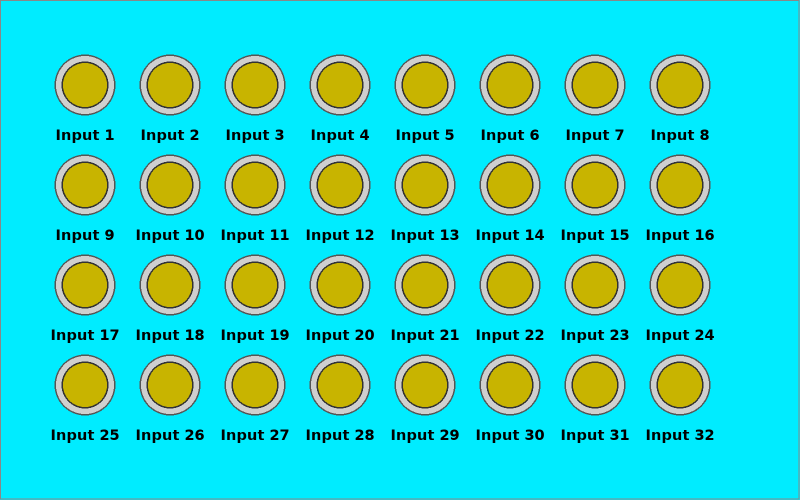
VISUALIZATION Screen_1_Sub_2  // 800x500
    Rectangle (0,0 800x500)
    Lamp1 (50,50 70x70), tooltip "Lamp 1", variable: GVL.HMI_Display_Lamp[0], style: Lamp-Lamp1-Yellow
    Label (50,120 70x30), "Input 1"
    Lamp1 (50,150 70x70), tooltip "Lamp 1", variable: GVL.HMI_Display_Lamp[8], style: Lamp-Lamp1-Yellow
    Label (50,220 70x30), "Input 9"
    Lamp1 (50,250 70x70), tooltip "Lamp 1", variable: GVL.HMI_Display_Lamp[16], style: Lamp-Lamp1-Yellow
    Label (50,320 70x30), "Input 17"
    Lamp1 (50,350 70x70), tooltip "Lamp 1", variable: GVL.HMI_Display_Lamp[24], style: Lamp-Lamp1-Yellow
    Label (50,420 70x30), "Input 25"
    Lamp1 (135,50 70x70), tooltip "Lamp 1", variable: GVL.HMI_Display_Lamp[1], style: Lamp-Lamp1-Yellow
    Label (135,120 70x30), "Input 2"
    Lamp1 (135,150 70x70), tooltip "Lamp 1", variable: GVL.HMI_Display_Lamp[9], style: Lamp-Lamp1-Yellow
    Label (135,220 70x30), "Input 10"
    Lamp1 (135,250 70x70), tooltip "Lamp 1", variable: GVL.HMI_Display_Lamp[17], style: Lamp-Lamp1-Yellow
    Label (135,320 70x30), "Input 18"
    Lamp1 (135,350 70x70), tooltip "Lamp 1", variable: GVL.HMI_Display_Lamp[25], style: Lamp-Lamp1-Yellow
    Label (135,420 70x30), "Input 26"
    Lamp1 (220,50 70x70), tooltip "Lamp 1", variable: GVL.HMI_Display_Lamp[2], style: Lamp-Lamp1-Yellow
    Label (220,120 70x30), "Input 3"
    Lamp1 (220,150 70x70), tooltip "Lamp 1", variable: GVL.HMI_Display_Lamp[10], style: Lamp-Lamp1-Yellow
    Label (220,220 70x30), "Input 11"
    Lamp1 (220,250 70x70), tooltip "Lamp 1", variable: GVL.HMI_Display_Lamp[18], style: Lamp-Lamp1-Yellow
    Label (220,320 70x30), "Input 19"
    Lamp1 (220,350 70x70), tooltip "Lamp 1", variable: GVL.HMI_Display_Lamp[26], style: Lamp-Lamp1-Yellow
    Label (220,420 70x30), "Input 27"
    Lamp1 (305,50 70x70), tooltip "Lamp 1", variable: GVL.HMI_Display_Lamp[3], style: Lamp-Lamp1-Yellow
    Label (305,120 70x30), "Input 4"
    Lamp1 (305,150 70x70), tooltip "Lamp 1", variable: GVL.HMI_Display_Lamp[11], style: Lamp-Lamp1-Yellow
    Label (305,220 70x30), "Input 12"
    Lamp1 (305,250 70x70), tooltip "Lamp 1", variable: GVL.HMI_Display_Lamp[19], style: Lamp-Lamp1-Yellow
    Label (305,320 70x30), "Input 20"
    Lamp1 (305,350 70x70), tooltip "Lamp 1", variable: GVL.HMI_Display_Lamp[27], style: Lamp-Lamp1-Yellow
    Label (305,420 70x30), "Input 28"
    Lamp1 (390,50 70x70), tooltip "Lamp 1", variable: GVL.HMI_Display_Lamp[4], style: Lamp-Lamp1-Yellow
    Label (390,120 70x30), "Input 5"
    Lamp1 (390,150 70x70), tooltip "Lamp 1", variable: GVL.HMI_Display_Lamp[12], style: Lamp-Lamp1-Yellow
    Label (390,220 70x30), "Input 13"
    Lamp1 (390,250 70x70), tooltip "Lamp 1", variable: GVL.HMI_Display_Lamp[20], style: Lamp-Lamp1-Yellow
    Label (390,320 70x30), "Input 21"
    Lamp1 (390,350 70x70), tooltip "Lamp 1", variable: GVL.HMI_Display_Lamp[28], style: Lamp-Lamp1-Yellow
    Label (390,420 70x30), "Input 29"
    Lamp1 (475,50 70x70), tooltip "Lamp 1", variable: GVL.HMI_Display_Lamp[5], style: Lamp-Lamp1-Yellow
    Label (475,120 70x30), "Input 6"
    Lamp1 (475,150 70x70), tooltip "Lamp 1", variable: GVL.HMI_Display_Lamp[13], style: Lamp-Lamp1-Yellow
    Label (475,220 70x30), "Input 14"
    Lamp1 (475,250 70x70), tooltip "Lamp 1", variable: GVL.HMI_Display_Lamp[21], style: Lamp-Lamp1-Yellow
    Label (475,320 70x30), "Input 22"
    Lamp1 (475,350 70x70), tooltip "Lamp 1", variable: GVL.HMI_Display_Lamp[29], style: Lamp-Lamp1-Yellow
    Label (475,420 70x30), "Input 30"
    Lamp1 (560,50 70x70), tooltip "Lamp 1", variable: GVL.HMI_Display_Lamp[6], style: Lamp-Lamp1-Yellow
    Label (560,120 70x30), "Input 7"
    Lamp1 (560,150 70x70), tooltip "Lamp 1", variable: GVL.HMI_Display_Lamp[14], style: Lamp-Lamp1-Yellow
    Label (560,220 70x30), "Input 15"
    Lamp1 (560,250 70x70), tooltip "Lamp 1", variable: GVL.HMI_Display_Lamp[22], style: Lamp-Lamp1-Yellow
    Label (560,320 70x30), "Input 23"
    Lamp1 (560,350 70x70), tooltip "Lamp 1", variable: GVL.HMI_Display_Lamp[30], style: Lamp-Lamp1-Yellow
    Label (560,420 70x30), "Input 31"
    Lamp1 (645,50 70x70), tooltip "Lamp 1", variable: GVL.HMI_Display_Lamp[7], style: Lamp-Lamp1-Yellow
    Label (645,120 70x30), "Input 8"
    Lamp1 (645,150 70x70), tooltip "Lamp 1", variable: GVL.HMI_Display_Lamp[15], style: Lamp-Lamp1-Yellow
    Label (645,220 70x30), "Input 16"
    Lamp1 (645,250 70x70), tooltip "Lamp 1", variable: GVL.HMI_Display_Lamp[23], style: Lamp-Lamp1-Yellow
    Label (645,320 70x30), "Input 24"
    Lamp1 (645,350 70x70), tooltip "Lamp 1", variable: GVL.HMI_Display_Lamp[31], style: Lamp-Lamp1-Yellow
    Label (645,420 70x30), "Input 32"
END_VISUALIZATION

(* stored: Version 1.1.0.1, ProductVersion 3.1.4024.12
   Visu Screen_1_Sub_2: Id {c5450f8c-8d7d-4238-aed7-2cd7db7f5009} *)
